PROGRAM ReadModbusCoils
VAR
	fbReadCoils       : FB_MBReadCoils;
    bReadCoils        : BOOL;
    bReadCoilsBusy    : BOOL;
    bReadCoilsError   : BOOL;
    nReadCoilsErrorId : UDINT;
    nReadCoilsCount   : UDINT;
    nQuantity         : WORD := 10;
    nMBAddr           : WORD := 32768;
    arrData           : ARRAY [0..1] OF BYTE;
	nTCPPort		  : UINT 	:= 502;
	nUnitID			  : BYTE	:= 255;
	tTimeout		  : TIME	:= T#1S;
END_VAR

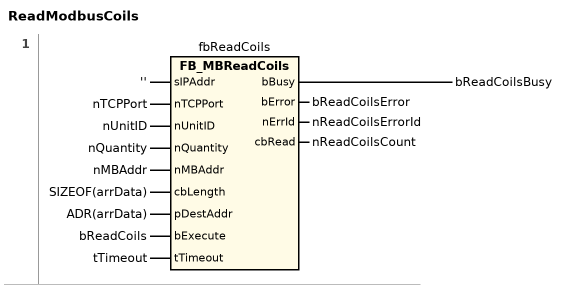
// NETWORK 1
fbReadCoils(
    sIPAddr := '',
    nTCPPort := nTCPPort,
    nUnitID := nUnitID,
    nQuantity := nQuantity,
    nMBAddr := nMBAddr,
    cbLength := SIZEOF(arrData),
    pDestAddr := ADR(arrData),
    bExecute := bReadCoils,
    tTimeout := tTimeout,
    bError => bReadCoilsError,
    nErrId => nReadCoilsErrorId,
    cbRead => nReadCoilsCount); // FB_MBReadCoils
bReadCoilsBusy := fbReadCoils.bBusy;

END_PROGRAM

(* stored: Version 1.1.0.1, ProductVersion 3.1.4024.12
   POU ReadModbusCoils: Id {de1a91fe-6c25-4214-b2cd-1da106c363a7}, SpecialFunc None *)
